Yaskawa INFORM job: KRIS2(-160_-90)34.JBI

/JOB
//NAME KRIS2(-160_-90)34
//POS
///NPOS 149,149,149,10,0,0
///TOOL 0
///POSTYPE PULSE
///PULSE
C00000=136908,-99459,-124829,-20670,71348,-76391
C00001=134470,-76528,-106815,-19279,71473,-77234
C00002=159578,-94739,-111578,-14965,102577,-71346
C00003=157566,-87256,-71357,-3912,80960,-68626
C00004=136911,-97837,-71335,-2043,74746,-75596
C00005=137353,-98864,-69097,-2107,72853,-75411
C00006=137353,-97788,-67030,-2113,72134,-75401
C00007=137490,-98681,-67551,-2126,71999,-75348
C00008=137823,-100474,-68178,-2166,71474,-75224
C00009=137490,-99527,-69160,-2120,72554,-75357
C00010=137490,-112967,-99500,-2043,84312,-75553
C00011=132962,-68022,-80970,-1616,95894,-77239
C00012=133097,-70190,-77189,-1618,92458,-77150
C00013=133258,-72060,-76849,-1633,91294,-77082
C00014=133258,-72050,-75890,-1633,90711,-77076
C00015=133258,-72054,-76082,-1633,90828,-77076
C00016=133486,-74582,-77287,-1655,90276,-76993
C00017=133258,-72036,-78289,-1635,92195,-77094
C00018=140979,-108094,-110643,-2385,93763,-74547
C00019=136708,-68987,-94400,-2043,103743,-76128
C00020=135283,-72263,-92514,-1875,100869,-76546
C00021=132985,-71970,-92089,-1645,100710,-77295
C00022=132985,-72383,-91264,-1643,99992,-77285
C00023=132985,-72300,-91437,-1643,100140,-77287
C00024=133184,-74834,-92632,-1655,99579,-77214
C00025=132985,-71000,-93741,-1657,102225,-77315
C00026=154221,-57088,-86668,-3768,105682,-70493
C00027=154636,-59803,-86532,-3777,104225,-70312
C00028=154636,-60502,-85461,-3758,103210,-70280
C00029=154636,-60414,-85604,-3761,103342,-70284
C00030=155113,-62506,-86695,-3797,102960,-70115
C00031=154600,-59756,-86288,-3773,104099,-70317
C00032=161369,-86849,-99090,-4273,98390,-67906
C00033=162299,-90705,-86659,-4280,88832,-67270
C00034=162680,-91589,-85702,-4311,87811,-67106
C00035=162680,-91368,-84537,-4311,87211,-67083
C00036=162680,-91407,-84732,-4311,87310,-67086
C00037=163568,-93888,-85727,-4385,86696,-66764
C00038=162680,-92039,-88633,-4311,89381,-67156
C00039=171854,-115132,-97044,-5055,83246,-63813
C00040=176135,-99923,-70409,-842,76306,-62354
C00041=176746,-100127,-69456,-876,75622,-62141
C00042=176746,-99180,-67670,-877,75010,-62140
C00043=176746,-99324,-67941,-877,75103,-62140
C00044=178145,-101177,-68585,-955,74562,-61655
C00045=175862,-99037,-69317,-825,76087,-62452
C00046=145436,-132582,-96247,390,75065,-72870
C00047=166235,-131980,-119843,-4599,88258,-65923
C00048=156260,-82084,-105550,-20461,72444,-69801
C00049=137260,-84248,-120477,-10166,77039,-76482
C00050=137260,-138866,-133764,-10166,31487,-76482
C00051=55958,-148097,-121035,-12961,13427,-75199
C00052=31464,-154695,-124663,-11622,10547,-75822
C00053=-11401,-148032,-125425,-11667,35640,-75771
C00054=-126225,-114648,-117375,-36487,17100,-65054
C00055=-160935,-140983,-109640,-13468,75088,-74332
C00056=-169853,-118963,-84593,-12681,69660,86771
C00057=-108998,-121589,-78490,3111,72246,67652
C00058=-101498,-120645,-75827,2941,70822,70188
C00059=-101498,-119392,-74038,2947,70366,70178
C00060=-101498,-119562,-74281,2946,70428,70180
C00061=-100817,-121900,-74755,2942,69496,70390
C00062=-101437,-120901,-75918,2941,70745,70208
C00063=-101671,-144527,-108100,2850,78408,70309
C00064=-107420,-98138,-90760,2968,91765,68662
C00065=-106123,-97431,-89210,2933,91127,69086
C00066=-106079,-97593,-88323,2932,90500,69086
C00067=-106079,-97314,-87194,2931,89950,69074
C00068=-106079,-97371,-87421,2931,90060,69077
C00069=-105757,-100151,-88472,2922,89269,69167
C00070=-106110,-97559,-89281,2933,91108,69092
C00071=-106110,-97729,-106489,3015,101600,69341
C00072=-107817,-77200,-97797,1990,101006,68606
C00073=-107961,-76698,-94617,1993,99314,68531
C00074=-107961,-77099,-93736,1989,98568,68519
C00075=-107961,-77014,-93933,1989,98733,68521
C00076=-107703,-80198,-95370,1956,97976,68594
C00077=-107832,-78083,-95841,1978,99355,68573
C00078=-108708,-76271,-95015,-4538,100749,88680
C00079=-108417,-78102,-94071,-4541,99246,88832
C00080=-149006,-93113,-100988,5479,101691,74295
C00081=-149599,-96300,-103483,5484,101628,74092
C00082=-108330,-77473,-93783,3039,98394,89923
C00083=-113965,-80387,-98246,3646,99862,88118
C00084=-112015,-122483,-114020,3369,87877,88431
C00085=-116962,-114728,-95357,3904,80614,86540
C00086=-117286,-114763,-93004,3949,79167,86382
C00087=-163022,-96736,-99152,-22139,103253,76925
C00088=-162158,-93804,-96763,-22109,103515,77196
C00089=-104767,-112354,-92165,2644,79373,90695
C00090=-109141,-112938,-93941,3100,80321,89215
C00091=-113958,-156480,-105404,3885,65233,87099
C00092=-113958,-135498,-81926,4007,61575,86972
C00093=-114943,-133176,-76806,4195,59669,86547
C00094=-163006,-94576,-83573,-21494,95359,78388
C00095=-162142,-91714,-81191,-21448,95589,78662
C00096=-98259,-129429,-76038,3501,60866,88602
C00097=-115088,-145817,-91151,6745,61908,86191
C00098=-120295,-145940,-91152,7309,62276,84335
C00099=-149731,-158641,-113843,-14975,70738,-69794
C00100=-149731,-158641,-113843,-14975,70738,-69794
C00101=-126225,-114648,-117375,-36487,17100,-65054
C00102=-118781,-153853,-134406,-32592,23357,-65054
C00103=-12470,-167083,-125425,-11667,16324,-75771
C00104=137258,-84249,-120477,-10166,64820,-76482
C00105=160540,-100857,-113063,-23155,68829,-67581
C00106=144636,-173309,-129138,-11293,64944,-72208
C00107=135566,-152591,-120530,-7709,74393,-76314
C00108=140848,-133584,-113559,-7137,84035,-75073
C00109=158743,-95268,-103371,-5812,102972,-69826
C00110=157888,-92366,-100981,-5813,102933,-70115
C00111=127361,-138532,-114921,-6064,81231,-79550
C00112=126467,-143470,-120820,-5933,82464,-79916
C00113=128645,-195873,-132590,-6758,63059,-78142
C00114=144821,-162395,-106929,-7940,65866,-72581
C00115=151353,-159653,-103782,-8374,65971,-70287
C00116=158755,-94787,-86481,976,103949,-69303
C00117=157900,-91912,-84097,841,103969,-69603
C00118=131040,-164995,-104643,-7049,61929,-77218
C00119=127169,-170980,-109668,-6701,61638,-78586
C00120=127203,-187747,-112013,-6590,55501,-77611
C00121=134083,-168892,-86258,5,48650,-76638
C00122=150686,-163778,-80153,-1742,47665,-70525
C00123=158782,-86330,-62292,-2348,97119,-70521
C00124=157926,-83586,-59872,-2521,97014,-70811
C00125=119290,-165255,-80160,-1845,46842,-81194
C00126=112444,-177354,-90291,-1803,46710,-83534
C00127=133031,-170450,-89431,9055,52143,-79525
C00128=147712,-143070,-77148,9897,64364,-73903
C00129=158743,-95268,-103371,-5812,102972,-69826
C00130=157888,-92366,-100981,-5813,102933,-70115
C00131=168512,-136452,-76172,10077,64775,-66770
C00132=153062,-184084,-115520,9876,66274,-71927
C00133=133135,-130401,-99458,8486,85928,-77222
C00134=133135,-130401,-99458,8486,85928,-77222
C00135=138110,-131166,-96474,8730,83193,-75716
C00136=158755,-94787,-86481,976,103949,-69303
C00137=157900,-91912,-84097,841,103969,-69603
C00138=151730,-125334,-94859,9131,83670,-71029
C00139=150058,-139901,-119688,9083,91560,-71028
C00140=133476,-138679,-117533,8523,92690,-76646
C00141=138175,-133983,-112919,8717,91763,-75095
C00142=158782,-86330,-62292,-2348,97119,-70521
C00143=157926,-83586,-59872,-2521,97014,-70811
C00144=149408,-127220,-110939,9086,92753,-71162
C00145=139154,-141635,-132500,8927,99684,-74194
C00146=159578,-94739,-111578,-14965,102577,-71346
C00147=134470,-76528,-106815,-19279,71473,-77234
C00148=36470,-76528,-106815,-19279,71473,-77234
BC00000=353519,332830,1075139
BC00001=353519,294132,1075139
BC00002=353519,214242,1075139
BC00003=382934,213120,1075139
BC00004=382934,213120,1075139
BC00005=382934,213120,1075139
BC00006=382934,213120,1075139
BC00007=382934,213120,1075136
BC00008=382934,213120,1075136
BC00009=382934,213120,1075136
BC00010=382934,213120,1075136
BC00011=382934,213120,1075136
BC00012=382934,213120,1075136
BC00013=382934,213120,1075136
BC00014=382934,213120,1075136
BC00015=382934,213120,1075136
BC00016=382934,213120,1075136
BC00017=382934,213120,1075136
BC00018=382076,183746,1075139
BC00019=382076,183746,1075139
BC00020=382076,183746,1075139
BC00021=382076,183746,1075139
BC00022=382076,183746,1075139
BC00023=382076,183746,1075139
BC00024=382076,183746,1075139
BC00025=382076,183746,1075139
BC00026=324696,183746,1075139
BC00027=324696,183746,1075139
BC00028=324696,183746,1075139
BC00029=324696,183746,1075139
BC00030=324696,183746,1075139
BC00031=324696,183746,1075139
BC00032=324696,183746,1075139
BC00033=324696,183746,1075139
BC00034=324696,183746,1075139
BC00035=324696,183746,1075139
BC00036=324696,183746,1075139
BC00037=324696,183746,1075139
BC00038=324696,183746,1075139
BC00039=324696,183746,1075139
BC00040=335320,183746,1075139
BC00041=335320,183746,1075139
BC00042=335320,183746,1075139
BC00043=335320,183746,1075139
BC00044=335320,183746,1075139
BC00045=335320,183746,1075139
BC00046=334019,183746,1075139
BC00047=382054,156718,1075139
BC00048=381880,223521,1075139
BC00049=353800,266120,1075139
BC00050=353800,266120,1075139
BC00051=373742,110742,1075139
BC00052=379757,63718,1075139
BC00053=398174,159824,1075139
BC00054=312616,52052,1075139
BC00055=340737,74809,1075139
BC00056=340750,75261,1075139
BC00057=340750,75261,1075135
BC00058=340750,75260,1075133
BC00059=340750,75260,1075133
BC00060=340750,75260,1075133
BC00061=340750,75260,1075133
BC00062=340750,75260,1075133
BC00063=340750,75260,1075133
BC00064=340750,75260,1075133
BC00065=340750,75260,1075133
BC00066=340750,75260,1075133
BC00067=340750,75260,1075133
BC00068=340750,75260,1075133
BC00069=340750,75260,1075133
BC00070=340750,75260,1075133
BC00071=340750,75260,1075133
BC00072=340750,75260,1075133
BC00073=340750,75260,1075133
BC00074=340750,75260,1075133
BC00075=340750,75260,1075133
BC00076=340750,75260,1075133
BC00077=340750,75260,1075133
BC00078=340750,75260,1075133
BC00079=340750,75260,1075133
BC00080=348896,99875,1075139
BC00081=348896,99875,1075139
BC00082=340750,75260,1075133
BC00083=340750,75260,1075133
BC00084=340750,75260,1075133
BC00085=340750,75260,1075133
BC00086=340750,75260,1075133
BC00087=322520,138659,1075139
BC00088=322520,138659,1075139
BC00089=340750,75260,1075133
BC00090=340750,75260,1075133
BC00091=340750,75260,1075133
BC00092=340750,75260,1075133
BC00093=340750,75260,1075133
BC00094=322446,111858,1075139
BC00095=322446,111858,1075139
BC00096=340750,75260,1075133
BC00097=340750,75260,1075133
BC00098=340750,75260,1075133
BC00099=340737,74809,1075139
BC00100=340737,74809,1075139
BC00101=312616,52052,1075139
BC00102=312616,52052,1075139
BC00103=398174,159824,1075139
BC00104=353801,266119,1075139
BC00105=381880,223521,1075139
BC00106=363620,145544,1075139
BC00107=363620,145544,1075139
BC00108=363620,145544,1075139
BC00109=364639,149103,1075139
BC00110=364639,149103,1075139
BC00111=363620,145544,1075139
BC00112=363923,145693,1075139
BC00113=363923,145693,1075139
BC00114=363923,145693,1075139
BC00115=363923,145693,1075139
BC00116=364758,151053,1075139
BC00117=364758,151053,1075139
BC00118=363923,145693,1075139
BC00119=363923,145693,1075139
BC00120=363923,145693,1075139
BC00121=363923,145693,1075139
BC00122=363923,145693,1075139
BC00123=355504,177664,1075139
BC00124=355504,177664,1075139
BC00125=363922,145691,1075138
BC00126=363923,145693,1075139
BC00127=304226,145693,1075139
BC00128=304226,145693,1075139
BC00129=364639,149103,1075139
BC00130=364639,149103,1075139
BC00131=304226,145693,1075139
BC00132=304226,145693,1075139
BC00133=304226,145693,1075139
BC00134=304226,145693,1075139
BC00135=304226,145693,1075139
BC00136=364758,151053,1075139
BC00137=364758,151053,1075139
BC00138=304226,145693,1075139
BC00139=304226,145693,1075139
BC00140=304226,124888,1075139
BC00141=304226,124888,1075139
BC00142=355504,177664,1075139
BC00143=355504,177664,1075139
BC00144=304226,124888,1075139
BC00145=304226,124888,1075139
BC00146=353519,214242,1075139
BC00147=353519,294132,1075139
BC00148=295309,515546,1075139
EC00000=1418945,372643
EC00001=1418945,372643
EC00002=1418945,372643
EC00003=1418945,372643
EC00004=1418945,372643
EC00005=1418945,372643
EC00006=1418945,372643
EC00007=1418944,372643
EC00008=1418944,372643
EC00009=1418944,372643
EC00010=1418944,372643
EC00011=1418944,372643
EC00012=1418944,372643
EC00013=1418944,372643
EC00014=1418944,372643
EC00015=1418944,372643
EC00016=1418944,372643
EC00017=1418944,372643
EC00018=1418945,372643
EC00019=1418945,372643
EC00020=1418945,372643
EC00021=1418945,372643
EC00022=1418945,372643
EC00023=1418945,372643
EC00024=1418945,372643
EC00025=1418945,372643
EC00026=1418945,372643
EC00027=1418945,372643
EC00028=1418945,372643
EC00029=1418945,372643
EC00030=1418945,372643
EC00031=1418945,372643
EC00032=1418945,372643
EC00033=1418945,372643
EC00034=1418945,372643
EC00035=1418945,372643
EC00036=1418945,372643
EC00037=1418945,372643
EC00038=1418945,372643
EC00039=1418945,372643
EC00040=1418945,372643
EC00041=1418945,372643
EC00042=1418945,372643
EC00043=1418945,372643
EC00044=1418945,372643
EC00045=1418945,372643
EC00046=1418945,372643
EC00047=1418945,372643
EC00048=1418945,372643
EC00049=1418945,372643
EC00050=1418945,372643
EC00051=1419033,372366
EC00052=1418945,372643
EC00053=1595090,-179995
EC00054=1773681,-740307
EC00055=1773681,-740307
EC00056=1773681,-740307
EC00057=1773682,-740305
EC00058=1773683,-740305
EC00059=1773683,-740305
EC00060=1773683,-740305
EC00061=1773683,-740305
EC00062=1773683,-740305
EC00063=1773683,-740305
EC00064=1773683,-740305
EC00065=1773683,-740305
EC00066=1773683,-740305
EC00067=1773683,-740305
EC00068=1773683,-740305
EC00069=1773683,-740305
EC00070=1773683,-740305
EC00071=1773683,-740305
EC00072=1773683,-740305
EC00073=1773683,-740305
EC00074=1773683,-740305
EC00075=1773683,-740305
EC00076=1773683,-740305
EC00077=1773683,-740305
EC00078=1773683,-740305
EC00079=1773683,-740305
EC00080=1773681,-740307
EC00081=1773681,-740307
EC00082=1773683,-740305
EC00083=1773683,-740305
EC00084=1773683,-740305
EC00085=1773683,-740305
EC00086=1773683,-740305
EC00087=1773681,-740307
EC00088=1773681,-740307
EC00089=1773683,-740305
EC00090=1773683,-740305
EC00091=1773683,-740305
EC00092=1773683,-740305
EC00093=1773683,-740305
EC00094=1773681,-740307
EC00095=1773681,-740307
EC00096=1773683,-740305
EC00097=1773683,-740305
EC00098=1773683,-740305
EC00099=1773681,-740307
EC00100=1773681,-740307
EC00101=1773681,-740307
EC00102=1773681,-740307
EC00103=1595090,-179995
EC00104=1418947,372636
EC00105=1418945,372643
EC00106=1418945,372643
EC00107=1418945,372643
EC00108=1418945,372643
EC00109=1418945,372643
EC00110=1418945,372643
EC00111=1418945,372643
EC00112=1418945,372643
EC00113=1418945,372643
EC00114=1418945,372643
EC00115=1418945,372643
EC00116=1418945,372643
EC00117=1418945,372643
EC00118=1418945,372643
EC00119=1418945,372643
EC00120=1418945,372643
EC00121=1418945,372643
EC00122=1418945,372643
EC00123=1418945,372643
EC00124=1418945,372643
EC00125=1418943,372641
EC00126=1418945,372643
EC00127=1418945,372643
EC00128=1418945,372643
EC00129=1418945,372643
EC00130=1418945,372643
EC00131=1418945,372643
EC00132=1418945,372643
EC00133=1418945,372643
EC00134=1418945,372643
EC00135=1418945,372643
EC00136=1418945,372643
EC00137=1418945,372643
EC00138=1418945,372643
EC00139=1418945,372643
EC00140=1418945,372643
EC00141=1418945,372643
EC00142=1418945,372643
EC00143=1418945,372643
EC00144=1418945,372643
EC00145=1418945,372643
EC00146=1418945,372643
EC00147=1418945,372643
EC00148=1418945,372643
///POSTYPE BASE
///RECTAN
///RCONF 0,0,0,0,1,0,0,0,0,0,0,0,0,0,0,0,0,0,0,0,0,0,0,0
P00006=2.006,1.622,-0.565,0.0000,0.0000,0.0000
P00021=0.073,2.058,-0.109,0.0000,0.0000,0.0000
P00022=2.006,1.622,-0.565,0.0000,0.0000,0.0000
///RCONF 0,0,0,0,0,0,0,0,0,0,0,0,0,0,0,0,0,0,0,0,0,0,0,0
P00023=-2.957,-4.083,2.762,0.0000,0.0000,0.0000
P00024=-1.466,-0.226,-0.419,0.0000,0.0000,0.0000
P00025=3.643,0.007,-2.585,0.0000,0.0000,0.0000
P00026=2.644,0.055,-2.583,0.0000,0.0000,0.0000
P00031=-0.170,0.039,-0.647,0.0000,0.0000,0.0000
P00032=-0.423,0.157,3.222,0.0000,0.0000,0.0000
P00033=0.854,-1.099,3.047,0.0000,0.0000,0.0000
//INST
///DATE 2024/12/19 16:40
///ATTR SC,RW
///GROUP1 RB1,BS1
///GROUP2 ST1
NOP
MOVJ C00000 BC00000 VJ=100.00  +MOVJ EC00000 VJ=100.00
MOVJ C00001 BC00001 VJ=100.00  +MOVJ EC00001 VJ=100.00
MOVJ C00002 BC00002 VJ=100.00  +MOVJ EC00002 VJ=100.00
'Path S1422
SFTOF3D
MOVJ C00003 BC00003 VJ=100.00  +MOVJ EC00003 VJ=100.00
MOVL C00004 BC00004 V=400.0  +MOVJ EC00004 VJ=100.00
SMOVL C00005 BC00005 V=100.0  +MOVJ EC00005
SREFP 3 C00006 BC00006  +REFP EC00006
CALL JOB:SEARCH-R1-S13D
SET P021 P006
SFTON3D P021
SMOVL C00007 BC00007 V=100.0  +MOVJ EC00007
SREFP 3 C00008 BC00008  +REFP EC00008
CALL JOB:SEARCH-R1-S13D
SET P021 P006
SFTON3D P021
SMOVL C00009 BC00009 V=100.0  +MOVJ EC00009
MOVL C00010 BC00010 V=400.0  +MOVJ EC00010 VJ=100.00
MOVL C00011 BC00011 V=1000.0  +MOVJ EC00011 VJ=100.00
MOVJ C00012 BC00012 VJ=100.00  +MOVJ EC00012 VJ=100.00
'Path S1423
SFTOF3D
SMOVL C00013 BC00013 V=100.0  +MOVJ EC00013
SREFP 3 C00014 BC00014  +REFP EC00014
CALL JOB:SEARCH-R1-S13D
SET P022 P006
SFTON3D P022
SMOVL C00015 BC00015 V=100.0  +MOVJ EC00015
SREFP 3 C00016 BC00016  +REFP EC00016
CALL JOB:SEARCH-R1-S13D
SET P022 P006
SFTON3D P022
SMOVL C00017 BC00017 V=100.0  +MOVJ EC00017
SFTOF3D
MOVL C00018 BC00018 V=400.0  +MOVJ EC00018 VJ=100.00
MOVL C00019 BC00019 V=1000.0  +MOVJ EC00019 VJ=100.00
MOVJ C00020 BC00020 VJ=100.00  +MOVJ EC00020 VJ=100.00
'Path S1424
SFTOF3D
SMOVL C00021 BC00021 V=100.0  +MOVJ EC00021
SREFP 3 C00022 BC00022  +REFP EC00022
CALL JOB:SEARCH-R1-S13D
SET P023 P006
SFTON3D P023
SMOVL C00023 BC00023 V=100.0  +MOVJ EC00023
SREFP 3 C00024 BC00024  +REFP EC00024
CALL JOB:SEARCH-R1-S13D
SET P023 P006
SFTON3D P023
SMOVL C00025 BC00025 V=100.0  +MOVJ EC00025
MOVL C00026 BC00026 V=400.0  +MOVJ EC00026 VJ=100.00
SMOVL C00027 BC00027 V=100.0  +MOVJ EC00027
SREFP 3 C00028 BC00028  +REFP EC00028
CALL JOB:SEARCH-R1-S13D
SET P024 P006
SFTON3D P024
SMOVL C00029 BC00029 V=100.0  +MOVJ EC00029
SREFP 3 C00030 BC00030  +REFP EC00030
CALL JOB:SEARCH-R1-S13D
SET P024 P006
SFTON3D P024
SMOVL C00031 BC00031 V=100.0  +MOVJ EC00031
MOVL C00032 BC00032 V=400.0  +MOVJ EC00032 VJ=100.00
MOVL C00033 BC00033 V=1000.0  +MOVJ EC00033 VJ=100.00
'Path S1423
SFTOF3D
SMOVL C00034 BC00034 V=100.0  +MOVJ EC00034
SREFP 3 C00035 BC00035  +REFP EC00035
CALL JOB:SEARCH-R1-S13D
SET P025 P006
SFTON3D P025
SMOVL C00036 BC00036 V=100.0  +MOVJ EC00036
SREFP 3 C00037 BC00037  +REFP EC00037
CALL JOB:SEARCH-R1-S13D
SET P025 P006
SFTON3D P025
SMOVL C00038 BC00038 V=100.0  +MOVJ EC00038
MOVL C00039 BC00039 V=400.0  +MOVJ EC00039 VJ=100.00
MOVL C00040 BC00040 V=1000.0  +MOVJ EC00040 VJ=100.00
'Path S1424
SFTOF3D
SMOVL C00041 BC00041 V=100.0  +MOVJ EC00041
SREFP 3 C00042 BC00042  +REFP EC00042
CALL JOB:SEARCH-R1-S13D
SET P026 P006
SFTON3D P026
SMOVL C00043 BC00043 V=100.0  +MOVJ EC00043
SREFP 3 C00044 BC00044  +REFP EC00044
CALL JOB:SEARCH-R1-S13D
SET P026 P006
SFTON3D P026
SFTOF3D
SMOVL C00045 BC00045 V=100.0  +MOVJ EC00045
MOVL C00046 BC00046 V=400.0  +MOVJ EC00046 VJ=100.00
MOVL C00047 BC00047 V=1000.0  +MOVJ EC00047 VJ=100.00
'obrot
MOVJ C00048 BC00048 VJ=100.00  +MOVJ EC00048 VJ=100.00
MOVJ C00049 BC00049 VJ=100.00  +MOVJ EC00049 VJ=100.00
MOVJ C00050 BC00050 VJ=100.00  +MOVJ EC00050 VJ=100.00
MOVJ C00051 BC00051 VJ=50.00  +MOVJ EC00051 VJ=50.00
MOVJ C00052 BC00052 VJ=100.00  +MOVJ EC00052 VJ=100.00
MOVJ C00053 BC00053 VJ=100.00  +MOVJ EC00053 VJ=100.00
MOVJ C00054 BC00054 VJ=100.00  +MOVJ EC00054 VJ=100.00
MOVJ C00055 BC00055 VJ=100.00  +MOVJ EC00055 VJ=100.00
'Path S1077
SFTOF3D
MOVJ C00056 BC00056 VJ=100.00  +MOVJ EC00056 VJ=100.00
MOVL C00057 BC00057 V=400.0  +MOVJ EC00057 VJ=100.00
SMOVL C00058 BC00058 V=100.0  +MOVJ EC00058
SREFP 3 C00059 BC00059  +REFP EC00059
CALL JOB:SEARCH-R1-S13D
SET P031 P006
SFTON3D P031
SMOVL C00060 BC00060 V=100.0  +MOVJ EC00060
SREFP 3 C00061 BC00061  +REFP EC00061
CALL JOB:SEARCH-R1-S13D
SET P031 P006
SFTON3D P031
SMOVL C00062 BC00062 V=100.0  +MOVJ EC00062
MOVL C00063 BC00063 V=1000.0  +MOVJ EC00063 VJ=100.00
MOVJ C00064 BC00064 VJ=100.00  +MOVJ EC00064 VJ=100.00
'Path S1078
SFTOF3D
MOVL C00065 BC00065 V=400.0  +MOVJ EC00065 VJ=100.00
SMOVL C00066 BC00066 V=100.0  +MOVJ EC00066
SREFP 3 C00067 BC00067  +REFP EC00067
CALL JOB:SEARCH-R1-S13D
SET P032 P006
SFTON3D P032
SMOVL C00068 BC00068 V=100.0  +MOVJ EC00068
SREFP 3 C00069 BC00069  +REFP EC00069
CALL JOB:SEARCH-R1-S13D
SET P032 P006
SFTON3D P032
SMOVL C00070 BC00070 V=100.0  +MOVJ EC00070
MOVL C00071 BC00071 V=1000.0  +MOVJ EC00071 VJ=100.00
'Path S1079
SFTOF3D
MOVL C00072 BC00072 V=400.0  +MOVJ EC00072 VJ=100.00
SMOVL C00073 BC00073 V=100.0  +MOVJ EC00073
SREFP 3 C00074 BC00074  +REFP EC00074
CALL JOB:SEARCH-R1-S13D
SET P033 P006
SFTON3D P033
SMOVL C00075 BC00075 V=100.0  +MOVJ EC00075
SREFP 3 C00076 BC00076  +REFP EC00076
CALL JOB:SEARCH-R1-S13D
SET P033 P006
SFTON3D P033
SMOVL C00077 BC00077 V=100.0  +MOVJ EC00077
SMOVL C00078 BC00078 V=166.7  +MOVJ EC00078
SFTON3D P033
SMOVL C00079 BC00079 V=133.3 PL=0  +MOVJ EC00079
SREFP 1 C00080 BC00080  +REFP EC00080
SREFP 2 C00081 BC00081  +REFP EC00081
MACRO1 MJ#(0) ARGF14
ARCON
SMOVL C00082 BC00082 V=10.0  +MOVJ EC00082
ARCOF
SMOVL C00083 BC00083 V=400.0  +MOVJ EC00083
SMOVL C00084 BC00084 V=1000.0  +MOVJ EC00084
SFTOF3D
MOVJ C00085 BC00085 VJ=100.00  +MOVJ EC00085 VJ=100.00
'Path W261
SFTOF3D
SFTON3D P032
SMOVL C00086 BC00086 V=133.3 PL=0  +MOVJ EC00086
SREFP 1 C00087 BC00087  +REFP EC00087
SREFP 2 C00088 BC00088  +REFP EC00088
MACRO1 MJ#(0) ARGF14
ARCON
SMOVL C00089 BC00089 V=10.0  +MOVJ EC00089
ARCOF
SMOVL C00090 BC00090 V=400.0  +MOVJ EC00090
SMOVL C00091 BC00091 V=1000.0  +MOVJ EC00091
SFTOF3D
'Path W1083
SFTOF3D
SFTON3D P031
MOVJ C00092 BC00092 VJ=100.00  +MOVJ EC00092 VJ=100.00
SMOVL C00093 BC00093 V=133.3 PL=0  +MOVJ EC00093
SREFP 1 C00094 BC00094  +REFP EC00094
SREFP 2 C00095 BC00095  +REFP EC00095
MACRO1 MJ#(0) ARGF14
ARCON
SMOVL C00096 BC00096 V=10.0  +MOVJ EC00096
ARCOF
SMOVL C00097 BC00097 V=400.0  +MOVJ EC00097
SFTOF3D
MOVJ C00098 BC00098 VJ=100.00  +MOVJ EC00098 VJ=50.00
'obrot
MOVJ C00099 BC00099 VJ=100.00  +MOVJ EC00099 VJ=100.00
MOVJ C00100 BC00100 VJ=100.00  +MOVJ EC00100 VJ=100.00
MOVJ C00101 BC00101 VJ=100.00  +MOVJ EC00101 VJ=100.00
MOVJ C00102 BC00102 VJ=100.00  +MOVJ EC00102 VJ=100.00
MOVJ C00103 BC00103 VJ=100.00  +MOVJ EC00103 VJ=100.00
MOVJ C00104 BC00104 VJ=100.00  +MOVJ EC00104 VJ=100.00
MOVJ C00105 BC00105 VJ=100.00  +MOVJ EC00105 VJ=100.00
'Path W1425
SFTOF3D
SFTON3D P023
MOVJ C00106 BC00106 VJ=100.00  +MOVJ EC00106 VJ=100.00
SMOVL C00107 BC00107 V=166.7  +MOVJ EC00107
SMOVL C00108 BC00108 V=133.3 PL=0  +MOVJ EC00108
SREFP 1 C00109 BC00109  +REFP EC00109
SREFP 2 C00110 BC00110  +REFP EC00110
MACRO1 MJ#(0) ARGF14
ARCON
SMOVL C00111 BC00111 V=10.0  +MOVJ EC00111
ARCOF
SMOVL C00112 BC00112 V=400.0  +MOVJ EC00112
SMOVL C00113 BC00113 V=1000.0  +MOVJ EC00113
SFTOF3D
'Path W1426
SFTOF3D
SFTON3D P022
MOVJ C00114 BC00114 VJ=100.00  +MOVJ EC00114 VJ=100.00
SMOVL C00115 BC00115 V=133.3 PL=0  +MOVJ EC00115
SREFP 1 C00116 BC00116  +REFP EC00116
SREFP 2 C00117 BC00117  +REFP EC00117
MACRO1 MJ#(0) ARGF14
ARCON
SMOVL C00118 BC00118 V=10.0  +MOVJ EC00118
ARCOF
SMOVL C00119 BC00119 V=400.0  +MOVJ EC00119
SMOVL C00120 BC00120 V=1000.0  +MOVJ EC00120
SFTOF3D
'Path W1427
SFTOF3D
SFTON3D P021
MOVJ C00121 BC00121 VJ=100.00  +MOVJ EC00121 VJ=100.00
SMOVL C00122 BC00122 V=133.3 PL=0  +MOVJ EC00122
SREFP 1 C00123 BC00123  +REFP EC00123
SREFP 2 C00124 BC00124  +REFP EC00124
MACRO1 MJ#(0) ARGF14
ARCON
SMOVL C00125 BC00125 V=10.0  +MOVJ EC00125
ARCOF
SMOVL C00126 BC00126 V=400.0  +MOVJ EC00126
SMOVL C00127 BC00127 V=166.7  +MOVJ EC00127
SFTON3D P026
SMOVL C00128 BC00128 V=133.3 PL=0  +MOVJ EC00128
SREFP 1 C00129 BC00129  +REFP EC00129
SREFP 2 C00130 BC00130  +REFP EC00130
MACRO1 MJ#(0) ARGF14
ARCON
SMOVL C00131 BC00131 V=10.0  +MOVJ EC00131
ARCOF
SMOVL C00132 BC00132 V=400.0  +MOVJ EC00132
SMOVL C00133 BC00133 V=1000.0  +MOVJ EC00133
SFTOF3D
'Path W1426
SFTOF3D
SFTON3D P025
MOVJ C00134 BC00134 VJ=100.00  +MOVJ EC00134 VJ=100.00
SMOVL C00135 BC00135 V=133.3 PL=0  +MOVJ EC00135
SREFP 1 C00136 BC00136  +REFP EC00136
SREFP 2 C00137 BC00137  +REFP EC00137
MACRO1 MJ#(0) ARGF14
ARCON
SMOVL C00138 BC00138 V=10.0  +MOVJ EC00138
ARCOF
SMOVL C00139 BC00139 V=400.0  +MOVJ EC00139
SMOVL C00140 BC00140 V=1000.0  +MOVJ EC00140
SFTOF3D
'Path W1427
SFTOF3D
SFTON3D P024
SMOVL C00141 BC00141 V=133.3 PL=0  +MOVJ EC00141
SREFP 1 C00142 BC00142  +REFP EC00142
SREFP 2 C00143 BC00143  +REFP EC00143
MACRO1 MJ#(0) ARGF14
ARCON
SMOVL C00144 BC00144 V=10.0  +MOVJ EC00144
ARCOF
SMOVL C00145 BC00145 V=400.0  +MOVJ EC00145
SFTOF3D
MOVJ C00146 BC00146 VJ=100.00  +MOVJ EC00146 VJ=100.00
MOVJ C00147 BC00147 VJ=100.00  +MOVJ EC00147 VJ=100.00
MOVJ C00148 BC00148 VJ=100.00  +MOVJ EC00148 VJ=100.00
END
